{attribute 'qualified_only'}
VAR_GLOBAL
	fbStart									: FB_Przycisk_NO;	//przycisk start
	fbStop									: FB_Przycisk_NO;	//przycisk stop
	fbWieza									: FB_WiezaSygnalizacyjna_Cyfrowe;	
	bUkladSafetyOK							: BOOL;
	bWcisnietyGrzyb							: ARRAY [1..10] OF BOOL;
//glowna metoda sterujaca
	fbSterowanieMaszyna						: FB_Sterowanie (	
															fbStart						:= fbStart,
													        fbStop						:= fbStop,
	                                                        fbWieza						:= fbWieza,
	                                                        bUkladSafetyOK				:= bUkladSafetyOK,
	                                                        bWcisnietyGrzyb				:= bWcisnietyGrzyb,
															iIloscGrzybowNaMaszynie		:= 1);
	
END_VAR

(* stored: Version 1.1.0.1, ProductVersion 3.1.4024.11
   GVL GVL_Sterowanie: Id {9ed956b7-beab-433c-bbb9-26959367f620} *)
